// TIA Portal V16 export
// export: Created 2023-08-28T09:37:52.8217437Z, ExportSetting WithDefaults, DisplayName Totally Integrated Automation Portal, DisplayVersion V16 Update 6, DisplayName TIA Portal Version Control Interface, DisplayVersion V16 Update 2, DisplayName TIA Portal Openness, DisplayVersion V16 Update 6, DisplayName STEP 7 Professional, DisplayVersion V16 Update 6, DisplayName STEP 7 Safety, DisplayVersion V16, DisplayName WinCC Advanced, DisplayVersion V16 Update 6
DATA_BLOCK "alarm_min_DN500_B5_DB"   // DB19
AUTHOR : rt69
VERSION : 0.1
// stored: AutoNumber true, DBAccessibleFromOPCUA true, InstanceOfName 01_E_Alarm_min_bar_empty_tanks, InstanceOfType FB
"01_E_Alarm_min_bar_empty_tanks"
   // VAR_OUTPUT
   //    bit_alarm_magistrala_min { ExternalAccessible := 'False'; ExternalVisible := 'False'; ExternalWritable := 'False'} : Bool;
   // END_VAR
   // VAR_IN_OUT
   //    bit_off_alarm_niskie_magistrala { ExternalAccessible := 'False'; ExternalVisible := 'False'; ExternalWritable := 'False'} : Bool;
   //    "tempStrategia Pompownia" : Int;
   //    "actStrategia Pompownia" : Int;
   // END_VAR
   // VAR
   //    memTriger_Strategia { ExternalAccessible := 'False'; ExternalVisible := 'False'; ExternalWritable := 'False'} : Bool;
   //    bit_normalne_magistrala { ExternalAccessible := 'False'; ExternalVisible := 'False'; ExternalWritable := 'False'} : Bool;
   //    bit_niskie_magistrala { ExternalAccessible := 'False'; ExternalVisible := 'False'; ExternalWritable := 'False'} : Bool;
   //    memFalling_allarm : Bool;
   // END_VAR
BEGIN
END_DATA_BLOCK
